FUNCTION_BLOCK EL2602
VAR
	{attribute addProperty Name "WcState"}
	_wcState : WcStateBase;
	{attribute addProperty Name "Info data"}
	_infoData : InfoDataBase;
	_io : EL2xx2_Data;
END_VAR

PROPERTY IO : REFERENCE TO EL2xx2_Data
GET
IO REF= _io;
END_GET
END_PROPERTY

PROPERTY WcState : REFERENCE TO WcStateBase
GET
WcState REF= _wcState;
END_GET
END_PROPERTY

END_FUNCTION_BLOCK

(* stored: Version 1.1.0.1, ProductVersion 3.1.4024.9
   POU EL2602: Id {84f6ee0e-e8f9-0a71-0154-5443fde65b09}, SpecialFunc None
   Property IO: Id {6e8aa94c-f227-02e7-27b6-28b6d32683ff}
   Get Get: Id {681d78c2-57bf-00e6-2cf6-250f267a97db}
   Property WcState: Id {4b56d4e9-bd47-0eff-11ec-a51ccdb23fe5}
   Get Get: Id {470df8d4-9701-0913-30f1-ec8e7080135a} *)
